(* Logix 5000 project; controller WWTP_SOLIDS_CLX vendor 1 type 14 code 54 rev 17.2; software revision 17.00; part 12 of 16 *)
(* tags used below, declared in another part *)
   Wrk_FirstColdStartT : TIMER;   // Time since first cold start
   Wrk_FirstFailColdT : TIMER;   // Time for cold motor to wait after 1st start failure before ready
   Wrk_SubsFailColdT : TIMER;   // Time for cold motor to wait after 2nd and subs. failures before ready
   Wrk_FirstFailHotT : TIMER;   // Time for hot motor to wait after 1st start failure before ready
   Wrk_SubsFailHotT : TIMER;   // Time for hot motor to wait after 2nd and subs. failures before ready
   Wrk_HotRestartOKT : TIMER;   // Time for hot motor to run so it can restart immediately when stopped
   Wrk_RestartHotT : TIMER;   // Time for hot motor to wait after stop after running less than Hot Restart OK time
   Wrk_HotToColdT : TIMER;   // Time for a stopped hot motor to become cold
   Wrk_State : DINT;   // Instruction State (see state diagram in design docs)
   Wrk_SecondColdStartT : TIMER;   // Time since second cold start
(* P_ResInh, continued *)

ROUTINE Prescan   (* ladder *)
// Clear timers and set to known state
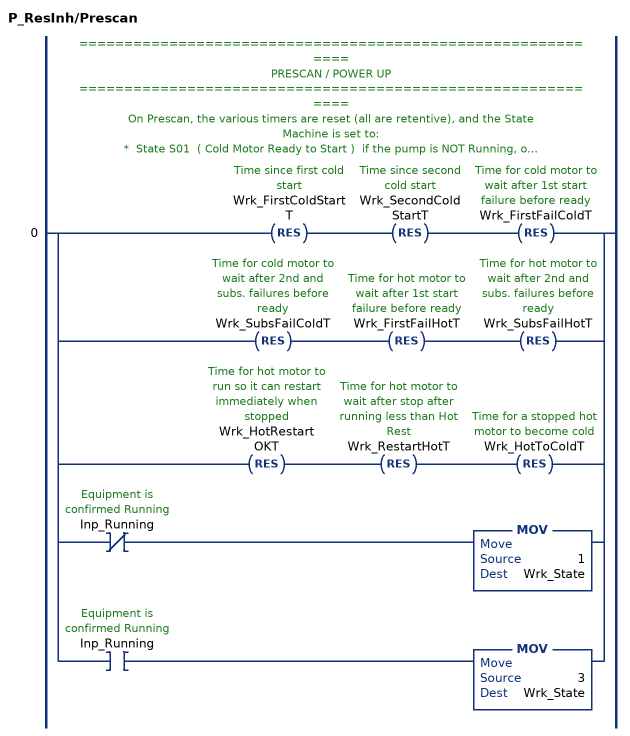
   // ============================================================
   // PRESCAN / POWER UP
   // ============================================================
   // On Prescan, the various timers are reset (all are retentive), and the State
   // Machine is set to:
   // *  State S01  ( Cold Motor Ready to Start )  if the pump is NOT Running, or
   // *  State S03  ( Cold Motor Running )  if the pump is Running.
   0: [RES(Wrk_FirstColdStartT) RES(Wrk_SecondColdStartT) RES(Wrk_FirstFailColdT) ,RES(Wrk_SubsFailColdT) RES(Wrk_FirstFailHotT) RES(Wrk_SubsFailHotT) ,RES(Wrk_HotRestartOKT) RES(Wrk_RestartHotT) RES(Wrk_HotToColdT) ,XIO(Inp_Running) MOV(1,Wrk_State) ,XIC(Inp_Running) MOV(3,Wrk_State) ];
END_ROUTINE
END_ADD_ON_INSTRUCTION

ADD_ON_INSTRUCTION P_RunTime   (* revision 0.7, ExecutePrescan, ExecuteEnableInFalse *)
// Run Time and Starts
// Revision note:
// Aligned name, description and local STRING values, sizes, across instructions.
// Help:
// This Instruction monitors the "Running" and "Starting" Status of a motor or other device and  provides:
// *  Total accumulated run time, in 1/10 hour increments (hour meter)
// *  Total number of starts or start attemptes (count)
// *  Maximum continuous run time for any start (hours)
// *  Program and Maintenance Commands to allow clearing of the totals/maximum
VAR_INPUT
   Inp_Starting : BOOL; {visible}   // 1=Motor is Starting (from motor instruction)
   Inp_Running : BOOL := 1; {visible}   // 1=Motor is Running (from motor instruction)
   Cfg_PCmdClear : BOOL := 1;   // 1=Clear Program Commands on receipt 0=Leave Set
   PCmd_ClearStarts : BOOL;   // Program Command to Clear Count of Starts (attempts)
   PCmd_ClearMaxHrs : BOOL;   // Program Command to Clear Maximum (continuous) Run Time for any start
   PCmd_ClearTotHrs : BOOL;   // Program Command to Clear Total Running Time
   MCmd_ClearStarts : BOOL;   // Maintenance Command to Clear Count of Starts (attempts)
   MCmd_ClearMaxHrs : BOOL;   // Maintenance Command to Clear Maximum (continuous) Run Time for any start
   MCmd_ClearTotHrs : BOOL;   // Maintenance Command to Clear Total Running Time
END_VAR
VAR_OUTPUT
   Val_Starts : DINT; {visible}   // Total number of motor starts or attempts
   Val_CurRunHrs : REAL; {visible}   // Current running time this start (hours)
   Val_MaxRunHrs : REAL; {visible}   // Maximum continuous running time for a given start (hours)
   Val_TotRunHrs : REAL; {visible}   // Total accumulated running time (hours)
END_VAR
VAR
   Wrk_CurHours : DINT;   // Whole hours of current run time
   Wrk_CurRunT : TIMER := (PRE := 2147483647);   // Timer for timing current run time
   Wrk_TotTenths : DINT;   // Tenths of hours of total run time
   Wrk_Starts : COUNTER := (PRE := 2147483647);   // Counter for counting motor starts
   Wrk_TotRunT : TIMER := (PRE := 2147483647);   // Retentive timer for timing 0.1 hour total run time
   Wrk_MaxHours : REAL;   // Internal Maximum Run Hours
END_VAR

ROUTINE EnableInFalse   (* ladder *)
// False Rung or Enable In False: as if motor is Stopped
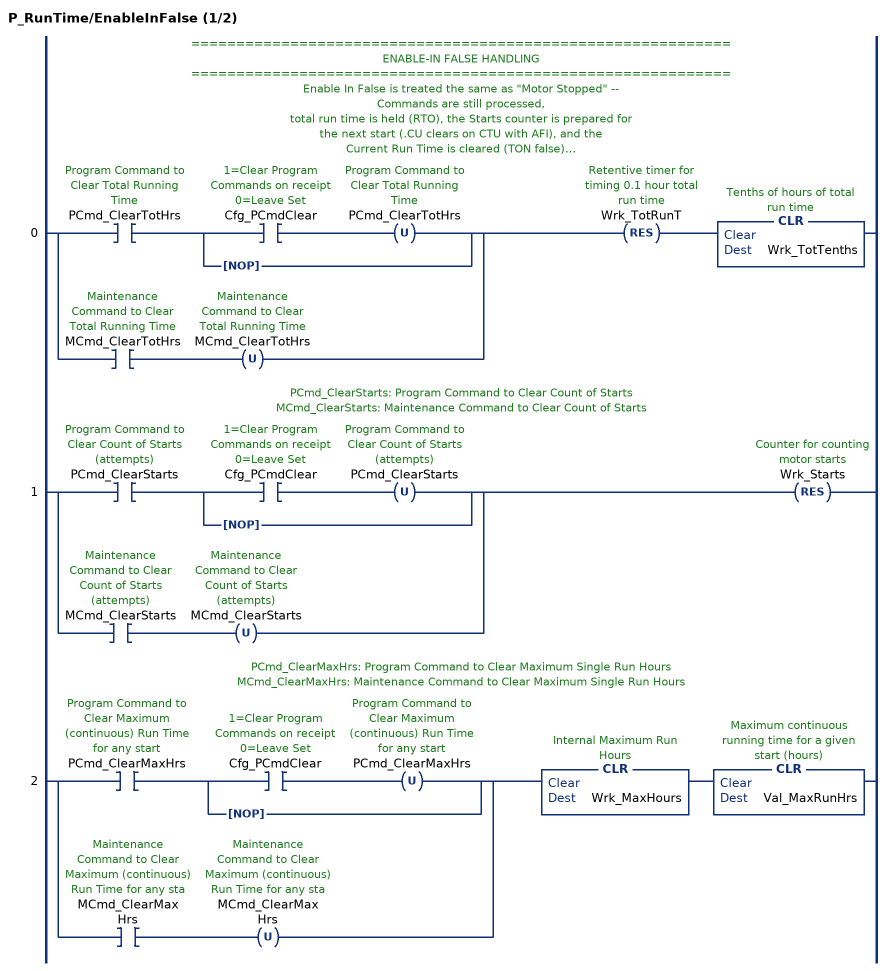
   // ============================================================
   // ENABLE-IN FALSE HANDLING
   // ============================================================
   // Enable In False is treated the same as "Motor Stopped" --
   // Commands are still processed,
   // total run time is held (RTO), the Starts counter is prepared for
   // the next start (.CU clears on CTU with AFI), and the
   // Current Run Time is cleared (TON false).
   // ============================================================
   // COMMAND PROCESSING
   // ============================================================
   // These rungs handle received Commands.  This object has no Modes and
   // Commands are accepted regardless of Mode.  Commands should be
   // restricted to authorized personnel (typically at a maintenance level).
   // PCmd_ClearTotHrs: Program Command to Clear Total Runtime Hours
   // MCmd_ClearTotHrs: Maintenance Command to Clear Total Runtime Hours
   0: [XIC(PCmd_ClearTotHrs) [XIC(Cfg_PCmdClear) OTU(PCmd_ClearTotHrs) ,NOP() ] ,XIC(MCmd_ClearTotHrs) OTU(MCmd_ClearTotHrs) ]RES(Wrk_TotRunT)CLR(Wrk_TotTenths);
   // PCmd_ClearStarts: Program Command to Clear Count of Starts
   // MCmd_ClearStarts: Maintenance Command to Clear Count of Starts
   1: [XIC(PCmd_ClearStarts) [XIC(Cfg_PCmdClear) OTU(PCmd_ClearStarts) ,NOP() ] ,XIC(MCmd_ClearStarts) OTU(MCmd_ClearStarts) ]RES(Wrk_Starts);
   // PCmd_ClearMaxHrs: Program Command to Clear Maximum Single Run Hours
   // MCmd_ClearMaxHrs: Maintenance Command to Clear Maximum Single Run Hours
   2: [XIC(PCmd_ClearMaxHrs) [XIC(Cfg_PCmdClear) OTU(PCmd_ClearMaxHrs) ,NOP() ] ,XIC(MCmd_ClearMaxHrs) OTU(MCmd_ClearMaxHrs) ]CLR(Wrk_MaxHours)CLR(Val_MaxRunHrs);
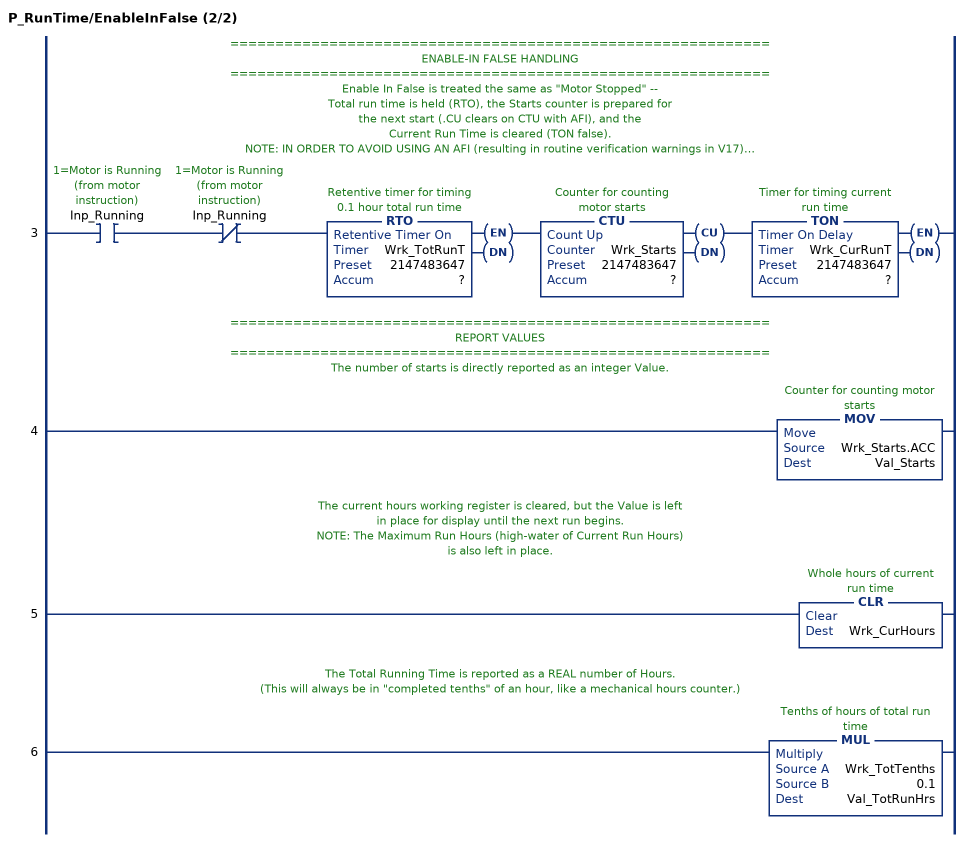
   // ============================================================
   // ENABLE-IN FALSE HANDLING
   // ============================================================
   // Enable In False is treated the same as "Motor Stopped" --
   // Total run time is held (RTO), the Starts counter is prepared for
   // the next start (.CU clears on CTU with AFI), and the
   // Current Run Time is cleared (TON false).
   // NOTE: IN ORDER TO AVOID USING AN AFI (resulting in routine verification warnings in V17),
   // THIS RUNG USES AN XIC AND XIO OF THE SAME BIT TO ENSURE THE
   // TIMERS AND COUNTER ARE SCANNED FALSE.
   // THIS IS NOT DEAD CODE.  IT IS INTENTIONALLY CODED THIS WAY FOR PROPER OPERATION.
   3: XIC(Inp_Running)XIO(Inp_Running)RTO(Wrk_TotRunT,?,?)CTU(Wrk_Starts,?,?)TON(Wrk_CurRunT,?,?);
   // ============================================================
   // REPORT VALUES
   // ============================================================
   // The number of starts is directly reported as an integer Value.
   4: MOV(Wrk_Starts.ACC,Val_Starts);
   // The current hours working register is cleared, but the Value is left
   // in place for display until the next run begins.
   // NOTE: The Maximum Run Hours (high-water of Current Run Hours)
   // is also left in place.
   5: CLR(Wrk_CurHours);
   // The Total Running Time is reported as a REAL number of Hours.
   // (This will always be in "completed tenths" of an hour, like a mechanical hours counter.)
   6: MUL(Wrk_TotTenths,0.1,Val_TotRunHrs);
END_ROUTINE

ROUTINE Logic   (* ladder *)
// Accumulate Run Time (if runnings) and Count Starts
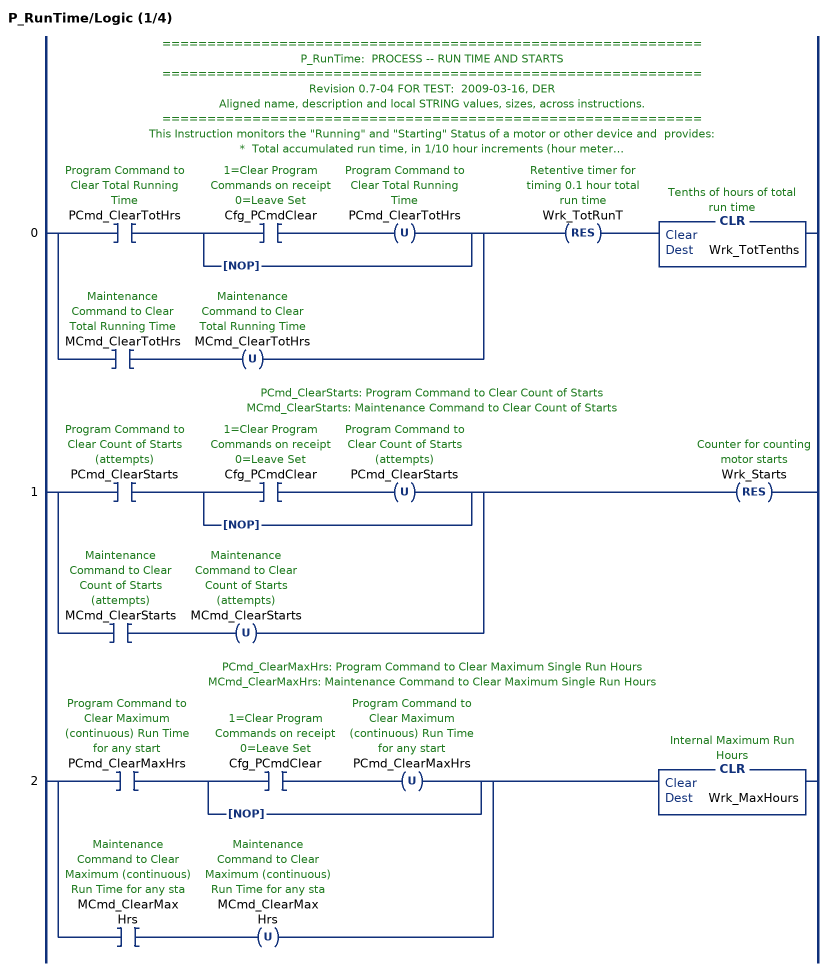
   // ============================================================
   // P_RunTime:  PROCESS -- RUN TIME AND STARTS
   // ============================================================
   // Revision 0.7-04 FOR TEST:  2009-03-16, DER
   // Aligned name, description and local STRING values, sizes, across instructions.
   // ============================================================
   // This Instruction monitors the "Running" and "Starting" Status of a motor or other device and  provides:
   // *  Total accumulated run time, in 1/10 hour increments (hour meter)
   // *  Total number of starts or start attemptes (count)
   // *  Maximum continuous run time for any start (hours)
   // * Commands to allow clearing of the totals/maximum
   // ============================================================
   // COMMAND PROCESSING
   // ============================================================
   // These rungs handle received Commands.  This object has no Modes and
   // Commands are accepted regardless of Mode.  Commands should be
   // restriceted to authorized personnel (typically at a maintenance level).
   // PCmd_ClearTotHrs: Program Command to Clear Total Runtime Hours
   // MCmd_ClearTotHrs: Maintenance Command to Clear Total Runtime Hours
   0: [XIC(PCmd_ClearTotHrs) [XIC(Cfg_PCmdClear) OTU(PCmd_ClearTotHrs) ,NOP() ] ,XIC(MCmd_ClearTotHrs) OTU(MCmd_ClearTotHrs) ]RES(Wrk_TotRunT)CLR(Wrk_TotTenths);
   // PCmd_ClearStarts: Program Command to Clear Count of Starts
   // MCmd_ClearStarts: Maintenance Command to Clear Count of Starts
   1: [XIC(PCmd_ClearStarts) [XIC(Cfg_PCmdClear) OTU(PCmd_ClearStarts) ,NOP() ] ,XIC(MCmd_ClearStarts) OTU(MCmd_ClearStarts) ]RES(Wrk_Starts);
   // PCmd_ClearMaxHrs: Program Command to Clear Maximum Single Run Hours
   // MCmd_ClearMaxHrs: Maintenance Command to Clear Maximum Single Run Hours
   2: [XIC(PCmd_ClearMaxHrs) [XIC(Cfg_PCmdClear) OTU(PCmd_ClearMaxHrs) ,NOP() ] ,XIC(MCmd_ClearMaxHrs) OTU(MCmd_ClearMaxHrs) ]CLR(Wrk_MaxHours);
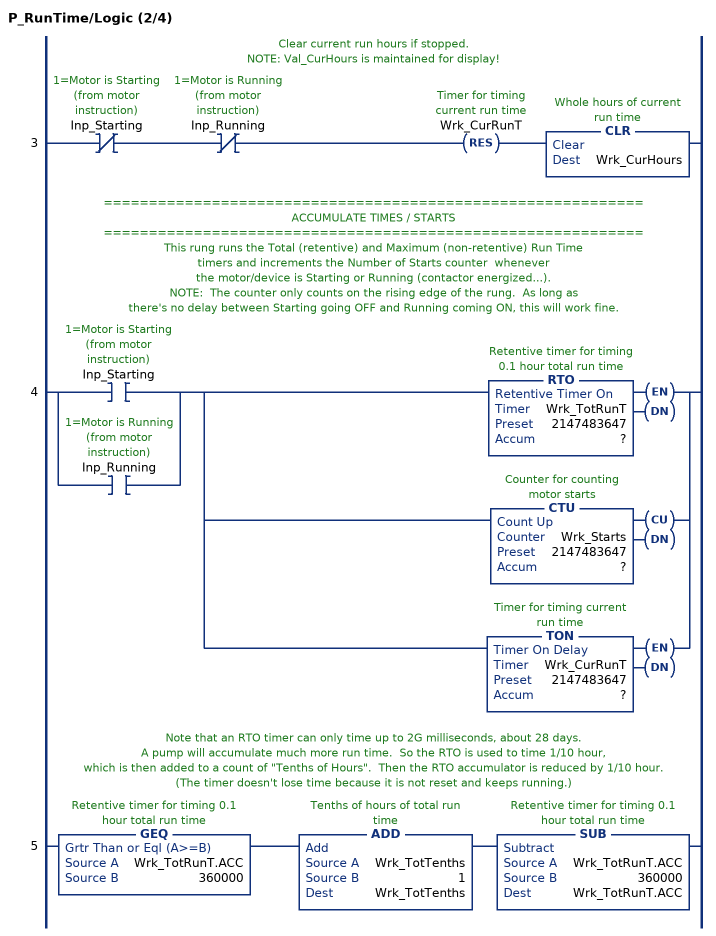
   // Clear current run hours if stopped.
   // NOTE: Val_CurHours is maintained for display!
   3: XIO(Inp_Starting)XIO(Inp_Running)RES(Wrk_CurRunT)CLR(Wrk_CurHours);
   // ============================================================
   // ACCUMULATE TIMES / STARTS
   // ============================================================
   // This rung runs the Total (retentive) and Maximum (non-retentive) Run Time
   // timers and increments the Number of Starts counter  whenever
   //  the motor/device is Starting or Running (contactor energized...).
   // NOTE:  The counter only counts on the rising edge of the rung.  As long as
   // there's no delay between Starting going OFF and Running coming ON, this will work fine.
   4: [XIC(Inp_Starting) ,XIC(Inp_Running) ][RTO(Wrk_TotRunT,?,?) ,CTU(Wrk_Starts,?,?) ,TON(Wrk_CurRunT,?,?) ];
   // Note that an RTO timer can only time up to 2G milliseconds, about 28 days.
   // A pump will accumulate much more run time.  So the RTO is used to time 1/10 hour,
   // which is then added to a count of "Tenths of Hours".  Then the RTO accumulator is reduced by 1/10 hour.
   // (The timer doesn't lose time because it is not reset and keeps running.)
   5: GEQ(Wrk_TotRunT.ACC,360000)ADD(Wrk_TotTenths,1,Wrk_TotTenths)SUB(Wrk_TotRunT.ACC,360000,Wrk_TotRunT.ACC);
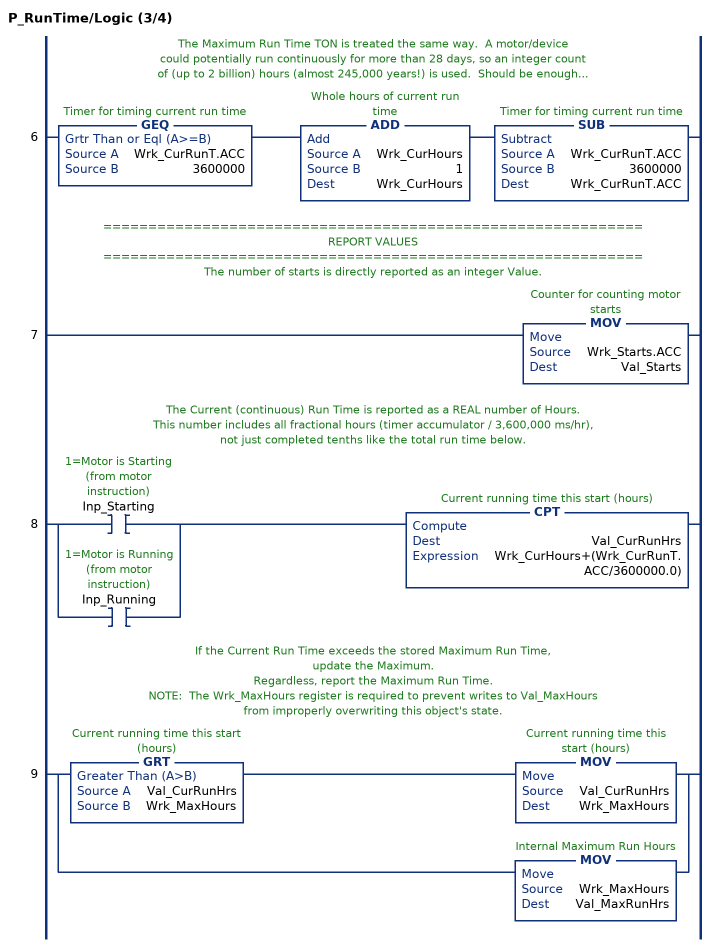
   // The Maximum Run Time TON is treated the same way.  A motor/device
   // could potentially run continuously for more than 28 days, so an integer count
   // of (up to 2 billion) hours (almost 245,000 years!) is used.  Should be enough...
   6: GEQ(Wrk_CurRunT.ACC,3600000)ADD(Wrk_CurHours,1,Wrk_CurHours)SUB(Wrk_CurRunT.ACC,3600000,Wrk_CurRunT.ACC);
   // ============================================================
   // REPORT VALUES
   // ============================================================
   // The number of starts is directly reported as an integer Value.
   7: MOV(Wrk_Starts.ACC,Val_Starts);
   // The Current (continuous) Run Time is reported as a REAL number of Hours.
   // This number includes all fractional hours (timer accumulator / 3,600,000 ms/hr),
   // not just completed tenths like the total run time below.
   8: [XIC(Inp_Starting) ,XIC(Inp_Running) ]CPT(Val_CurRunHrs,Wrk_CurHours+(Wrk_CurRunT.ACC/3600000.0));
   // If the Current Run Time exceeds the stored Maximum Run Time,
   // update the Maximum.
   // Regardless, report the Maximum Run Time.
   // NOTE:  The Wrk_MaxHours register is required to prevent writes to Val_MaxHours
   // from improperly overwriting this object's state.
   9: [GRT(Val_CurRunHrs,Wrk_MaxHours) MOV(Val_CurRunHrs,Wrk_MaxHours) ,MOV(Wrk_MaxHours,Val_MaxRunHrs) ];
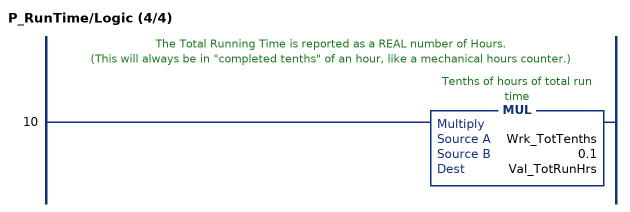
   // The Total Running Time is reported as a REAL number of Hours.
   // (This will always be in "completed tenths" of an hour, like a mechanical hours counter.)
   10: MUL(Wrk_TotTenths,0.1,Val_TotRunHrs);
END_ROUTINE

ROUTINE Prescan   (* ladder *)
// Set Current Run time internally to 0.  Display value is left in place.
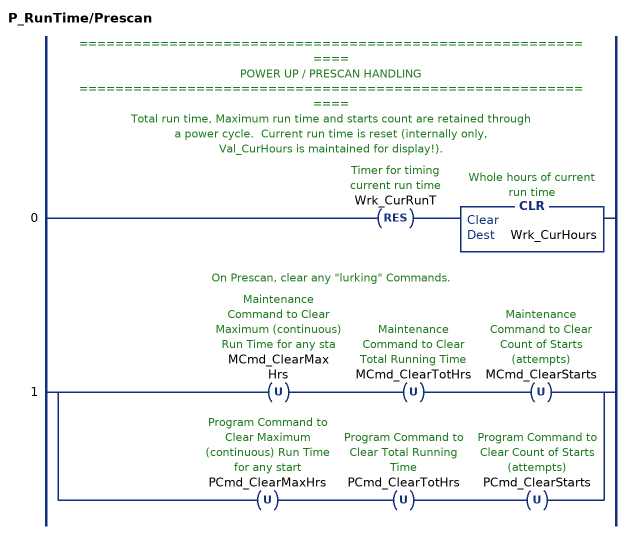
   // ============================================================
   // POWER UP / PRESCAN HANDLING
   // ============================================================
   // Total run time, Maximum run time and starts count are retained through
   // a power cycle.  Current run time is reset (internally only,
   // Val_CurHours is maintained for display!).
   0: RES(Wrk_CurRunT)CLR(Wrk_CurHours);
   // On Prescan, clear any "lurking" Commands.
   1: [OTU(MCmd_ClearMaxHrs) OTU(MCmd_ClearTotHrs) OTU(MCmd_ClearStarts) ,OTU(PCmd_ClearMaxHrs) OTU(PCmd_ClearTotHrs) OTU(PCmd_ClearStarts) ];
END_ROUTINE
END_ADD_ON_INSTRUCTION

ADD_ON_INSTRUCTION P_ValveMO   (* revision 0.9, ExecutePrescan, ExecuteEnableInFalse *)
// Motor Operated Valve
// Revision note:
// Aligned name, description and local STRING values, sizes, across instructions.
// Help:
// This Instruction controls and monitors a motor-operated
// valve (typ. two position: opened, closed) and provides:
// *  Ability to command valve to open, command valve to close, and,
//      optionally, command valve to stop motion (operator only)
// *  Ability to reverse valve travel (for valves with the ability to accept a Stop output)
// *  Monitoring of limit switch feedback, display of actual valve status
// *  Detection of failure to move (full stall), failure to reach position (transit stall)
// *  Monitoring of Permissive conditions to motor the valve open, and separate
//      Permissive conditions to motor the valve closed
// *  Simulation, providing feedback of a working valve while disabling outputs
// *  Monitoring of I/O communication faults
// *  Alarms for Full Stall, Transit Stall, Actuator Failure (separate input), I/O Fault
// *  Operation in Hand, Maintenance, Override, Program and Operator Modes
// *  "Available" status for use by automation logic to know whether valve
//      can be controlled by other objects.
VAR_INPUT
   Inp_OpenLS : BOOL; {visible}   // Valve Open Limit Switch 1=confirmed OPEN
   Inp_ClosedLS : BOOL; {visible}   // Valve Closed Limit Switch 1=confirmed CLOSED
   Inp_ActuatorFault : BOOL; {visible}   // Valve Actuator Fault (overload, etc.), 0=OK, 1=Fault)
   Inp_OpenPermOK : BOOL := 1; {visible}   // 1=Open Permissives OK, Valve can motor open
   Inp_OpenNBPermOK : BOOL := 1; {visible}   // 1=Non-Bypassable Open Permissives OK, valve can motor open
   Inp_ClosePermOK : BOOL := 1; {visible}   // 1=Close Permissives OK, Valve can motor closed
   Inp_CloseNBPermOK : BOOL := 1; {visible}   // 1=Non-Bypassable Close Permissives OK, valve can motor closed
   Inp_IOFault : BOOL;   // Input Communication Status 0=OK, 1=fail
   Inp_Sim : BOOL;   // 1=Simulate working valve; 0=Open/Close/ Monitor actual valve
   Inp_Hand : BOOL; {visible}   // 1=Select Hand (hardwired) Mode
   Inp_Ovrd : BOOL; {visible}   // 1=Select Override Mode
   Inp_OvrdOpen : BOOL; {visible}   // 1=Override to OPEN, 0=do not override open
   Inp_OvrdClose : BOOL; {visible}   // 1=Override to CLOSED, 0=do not override closed
   Inp_OvrdStop : BOOL;   // 1=Override to STOP moving, 0=do not override to STOP
   Inp_Reset : BOOL; {visible}   // 1=Reset all fault conditions and latched Alarms
   Cfg_HasOpenLS : BOOL;   // 1=Valve provides an Open Limit Switch signal
   Cfg_HasClosedLS : BOOL;   // 1=Valve provides a Closed Limit Switch signal
   Cfg_UseOpenLS : BOOL;   // 1=Valve Open LS should be used for failure checking
   Cfg_UseClosedLS : BOOL;   // 1=Valve Closed LS should be used for failure checking
   Cfg_LSFail : BOOL := 1;   // 1=both switches ON=fail, 0=both switches OFF=fail
   Cfg_HasStop : BOOL;   // 1=Stop output can be used to break local seal-in and stop valve motion
   Cfg_HasOpenPermObj : BOOL;   // 1=Tells HMI a P_Perm is connected to Inp_OpenPermOK
   Cfg_HasClosePermObj : BOOL;   // 1=Tells HMI a P_Perm is connected to Inp_ClosePermOK
   Cfg_PCmdClear : BOOL := 1;   // 1=Clear Program Commands on receipt 0=Leave Set
   Cfg_OvrdPerm : BOOL;   // 1=Override ignores Bypassable Perm; 0=always use Perm
   Cfg_HasFullStallAlm : BOOL;   // 1=Full Stall Alarm exists and will be checked
   Cfg_HasTransitStallAlm : BOOL;   // 1=Transit Stall Alarm exists and will be checked
   Cfg_HasActuatorFaultAlm : BOOL;   // 1=Actuator Fault Alarm exists and will be checked
   Cfg_HasIOFaultAlm : BOOL;   // 1=I/O Fault Alarm exists and will be checked
   Cfg_FullStallResetReqd : BOOL;   // 1=Reset requied to clear Full Stall Alarm
   Cfg_TransitStallResetReqd : BOOL;   // 1=Reset required to clear Transit Stall Alarm
   Cfg_ActuatorFaultResetReqd : BOOL;   // 1=Reset required to clear Actuator Fault Alarm
   Cfg_IOFaultResetReqd : BOOL;   // 1=Reset required to clear I/O Fault Alarm
   Cfg_FullStallAckReqd : BOOL := 1;   // 1=Acknowledge required for Full Stall Alarm
   Cfg_TransitStallAckReqd : BOOL := 1;   // 1=Acknowledge required for Transit Stall Alarm
   Cfg_ActuatorFaultAckReqd : BOOL := 1;   // 1=Acknowledge required for Actuator Fault Alarm
   Cfg_IOFaultAckReqd : BOOL := 1;   // 1=Acknowledge required for I/O Fault Alarm
   Cfg_FullStallSeverity : SINT := 4;   // Full Stall Alarm Severity 1=info 2=warn 3=excep 4=fault
   Cfg_TransitStallSeverity : SINT := 4;   // Transit Stall Alarm Severity 1=info 2=warn 3=excep 4=fault
   Cfg_ActuatorFaultSeverity : SINT := 2;   // Actuator Fault Alarm Severity 1=info 2=warn 3=excep 4=fault
   Cfg_IOFaultSeverity : SINT := 4;   // I/O Fault Alarm Severity 1=info 2=warn 3=excep 4=fault
   Cfg_OutPulseT : DINT := 5;   // Time (in seconds) to pulse valve outputs (0 = outputs maintained ON)
   Cfg_SimFdbkT : DINT := 20;   // Delay to echo back of Open/Closed status when in Simulation (sec)
   Cfg_FullStallT : DINT := 15;   // After commanded, time with no motion before Fault (sec)
   Cfg_TransitStallT : DINT := 60;   // After command, time to reach position before fault (sec)
   PSet_Owner : DINT;   // Program Owner Request ID (non-zero) or Release (zero)
   PCmd_Open : BOOL;   // Program Command to Open Valve
   PCmd_Close : BOOL;   // Program Command to Close Valve
   PCmd_Acq : BOOL;   // Program Command to Acquire ownership (Oper/OOS to Prog)
   PCmd_Rel : BOOL;   // Program Command to Release ownership (Prog to OOS)
   PCmd_Lock : BOOL;   // Program Command to Lock Mode in Prog
   PCmd_Unlock : BOOL;   // Program Command to Unlock Mode
   PCmd_Reset : BOOL;   // Program Command to Reset all Alarms requiring Reset
   PCmd_FullStallAck : BOOL;   // Program Command to Acknowledge Full Stall Alarm
   PCmd_FullStallInhibit : BOOL;   // Program Command to Inhibit Full Stall Alarm
   PCmd_FullStallUninhibit : BOOL;   // Program Command to Uninhibit Full Stall Alarm
   PCmd_TransitStallAck : BOOL;   // Program Command to Acknowledge Transit Stall Alarm
   PCmd_TransitStallInhibit : BOOL;   // Program Command to Inhibit Transit Stall Alarm
   PCmd_TransitStallUninhibit : BOOL;   // Program Command to Uninhibit Transit Stall Alarm
   PCmd_ActuatorFaultAck : BOOL;   // Program Command to Acknowledge Actuator Fault Alarm
   PCmd_ActuatorFaultInhibit : BOOL;   // Program Command to Inhibit Actuator Fault Alarm
   PCmd_ActuatorFaultUninhibit : BOOL;   // Program Command to Uninhibit Actuator Fault Alarm
   PCmd_IOFaultAck : BOOL;   // Program Command to Acknowledge I/O Fault Alarm
   PCmd_IOFaultInhibit : BOOL;   // Program Command to Inhibit I/O Fault Alarm
   PCmd_IOFaultUninhibit : BOOL;   // Program Command to Uninhibit I/O Fault Alarm
   OCmd_Open : BOOL;   // Operator Command to Open Valve
   OCmd_Close : BOOL;   // Operator Command to Close Valve
   OCmd_Stop : BOOL;   // Operator Command to Stop Valve Motion
   OCmd_Bypass : BOOL;   // Operator Command to Bypass all Bypassable Interlocks and Permissives
   OCmd_Check : BOOL;   // Operator Command to Check (not bypass) all Interlocks and Permissives
   MCmd_Disable : BOOL;   // Maintenance Command to Disable Valve
   MCmd_Enable : BOOL;   // Maintenance Command to Enable (allow to energize) Valve
   OCmd_Reset : BOOL;   // Operator Command to Reset all Alarms requiring Reset
END_VAR
VAR_OUTPUT
   Out_Open : BOOL; {visible}   // 1=Run actuator motor to OPEN Valve
   Out_Close : BOOL; {visible}   // 1=Run actuator motor to CLOSE Valve
   Out_Stop : BOOL;   // 1=Break seal-in circuit in actuator to STOP Valve motion
   Val_Owner : DINT;   // Current Object Owner ID (0=not owned)
   Val_Notify : SINT;   // Current Alarm Level and Acknowledgement (enumeration)
   Sts_Closed : BOOL; {visible}   // 1=Valve requested to Close and is confirmed Closed
   Sts_CmdToOpen : BOOL; {visible}   // 1=Valve commanded to Open, has not yet moved off Open LS
   Sts_Opening : BOOL; {visible}   // 1=Valve requested to open and awaiting open feedback
   Sts_Opened : BOOL; {visible}   // 1=Valve requested to open and is confirmed Opened
   Sts_CmdToClose : BOOL; {visible}   // 1=Valve commanded to Close, has not yet moved off Closed LS
   Sts_Closing : BOOL; {visible}   // 1=Valve requested to Close and awaiting Closed feedback
   Sts_Stopped : BOOL;   // 1=Valve requested to Stop and is not at either end of travel
   Sts_Available : BOOL;   // 1=Valve available for control by automation (Prog)
   Sts_Bypass : BOOL;   // 1=Bypassable Interlocks and Permissives are Bypassed
   Sts_Disabled : BOOL;   // 1=Valve is Disabled
   Sts_LSFail : BOOL;   // 1=Limit Switch Overlap Failure
   Sts_Err : BOOL; {visible}   // 1=Error in Config: see detail bits for reason
   Err_Timer : BOOL;   // 1=Error in Config: Invalid Check or Pulse Time (use 0 to 2147483)
   Err_Sim : BOOL;   // 1=Error in Config: Simulation timer preset (use 0 to 2147483)
   Err_Alarm : BOOL;   // 1=Error in Config: Invalid Alarm Severity
   Sts_Hand : BOOL; {visible}   // 1=Mode is Hand (supersedes Maint, Ovrd, Prog, Oper)
   Sts_Maint : BOOL; {visible}   // 1=Mode is Maintenance (supersedes Ovrd, Prog, Oper)
   Sts_Ovrd : BOOL; {visible}   // 1=Mode is Override (supersedes Prog, Oper)
   Sts_Prog : BOOL; {visible}   // 1=Mode is Program (auto)
   Sts_Oper : BOOL := 1; {visible}   // 1=Mode is Operator (manual)
   Sts_ProgOperLock : BOOL;   // 1=Program or Operator has requested Mode Lock
   Sts_FullStall : BOOL;   // 1=Valve Full Stall (failed to move at all) (One-Shot)
   Alm_FullStall : BOOL;   // 1=Valve Full Stall (failed to move at all) Alarm
   Ack_FullStall : BOOL;   // 1=Full Stall Alarm has been acknowledged
   Sts_FullStallDisabled : BOOL;   // 1=Full Stall Alarm has been disabled (will not be sent)
   Sts_FullStallInhibited : BOOL;   // 1=Full Stall Alarm has been inhibited by logic
   Sts_FullStallSuppressed : BOOL;   // 1=Full Stall Alarm has been suppressed (logged only)
   Sts_TransitStall : BOOL;   // 1=Valve Transit Stall (did not reach target position) (One-Shot)
   Alm_TransitStall : BOOL;   // 1=Valve Transit Stall (did not reach target pos.) Alarm
   Ack_TransitStall : BOOL;   // 1=Transit Stall Alarm has been acknowledged
   Sts_TransitStallDisabled : BOOL;   // 1=Transit Stall Alarm has been disabled (will not be sent)
   Sts_TransitStallInhibited : BOOL;   // 1=Transit Stall Alarm has been inhibited by logic
   Sts_TransitStallSuppressed : BOOL;   // 1=Transit Stall Alarm has been suppressed (logged only)
   Sts_ActuatorFault : BOOL;   // 1=Actuator Fault detected (input)
   Alm_ActuatorFault : BOOL;   // 1=Alarm: Actuator Fault Detected
   Ack_ActuatorFault : BOOL;   // 1=Actuator Fault Alarm has been acknowledged
   Sts_ActuatorFaultDisabled : BOOL;   // 1=Actuator Fault Alarm is Disabled (not saved or sent)
   Sts_ActuatorFaultInhibited : BOOL;   // 1=Actuator Fault Alarm has been inhibited by logic
   Sts_ActuatorFaultSuppressed : BOOL;   // 1=Actuator Fault Alarm has been suppressed (logged only)
   Sts_IOFault : BOOL;   // I/O Comm Fault Status (0=OK, 1=Bad)
   Alm_IOFault : BOOL;   // 1=I/O Fault Alarm
   Ack_IOFault : BOOL;   // 1=I/O Fault Alarm has been acknowledged
   Sts_IOFaultDisabled : BOOL;   // 1=I/O Fault Alarm is Disabled (not saved or sent)
   Sts_IOFaultInhibited : BOOL;   // 1=I/O Fault Alarm has been inhibited by logic
   Sts_IOFaultSuppressed : BOOL;   // 1=I/O Fault Alarm has been suppressed (logged only)
   Rdy_Open : BOOL;   // 1=Ready to receive OCmd_Open (enables HMI button)
   Rdy_Close : BOOL;   // 1=Ready to receive OCmd_Close (enables HMI button)
   Rdy_Stop : BOOL;   // 1=Ready to receive OCmd_Stop (enables HMI button)
   Rdy_Bypass : BOOL;   // 1=Ready to receive OCmd_Bypass (enables HMI button)
   Rdy_Check : BOOL;   // 1=Ready to receive OCmd_Check (enables HMI button)
   Rdy_Disable : BOOL;   // 1=Ready to receive MCmd_Disable (enables HMI button)
   Rdy_Enable : BOOL;   // 1=Ready to receive MCmd_Enable (enables HMI button)
   Rdy_Reset : BOOL;   // 1=Ready to receive OCmd_Reset (enables HMI button)
END_VAR
VAR
   Mode : P_Mode := (Cfg_PCmdClear := 1, Cfg_OvrdOverLock := 1, Sts_Oper := 1, Rdy_Rel := 1, Rdy_AcqLock := 1);   // Valve Mode Selection
   IOFault : P_Alarm := (Inp := 1, Cfg_AckReqd := 1, Cfg_Severity := 3, Ack := 1, Rdy_Disable := 1);   // I/O Fault Alarm
   ActuatorFault : P_Alarm := (Inp := 1, Cfg_AckReqd := 1, Cfg_Severity := 3, Ack := 1, Rdy_Disable := 1);   // Actuator Fault Alarm
   TransitStall : P_Alarm := (Inp := 1, Cfg_AckReqd := 1, Cfg_Severity := 3, Ack := 1, Rdy_Disable := 1);   // Valve Transit Stall (moved but did not reach target) Alarm
   FullStall : P_Alarm := (Inp := 1, Cfg_AckReqd := 1, Cfg_Severity := 3, Ack := 1, Rdy_Disable := 1);   // Valve Full Stall (did not move) Alarm
   Cfg_Tag : STRING_20 := 'P_ValveMO';   // Tagname for display on HMI
   Cfg_Label : STRING_20 := 'Valve Control';   // Label for graphic symbol displayed on HMI
   Cfg_Desc : STRING_40 := 'Motor Operated Valve';   // Description for display on HMI
   Wrk_Open : BOOL;   // 1=Requested to OPEN Valve
   Wrk_SimOpenT : TIMER;   // Simulation Delay until Opened
   Wrk_Fault : BOOL;   // 1=a Valve Fault has been detected
   Wrk_SimCloseT : TIMER;   // Simulation Delay until Closed
   Wrk_OpenFdbk : BOOL;   // 1=LS Feedback shows valve confirmed open
   Wrk_Notify : DINT;   // Buffer for building Val_Notify
   Wrk_Bypass : BOOL;   // Internal Bypassable Permissives and Interlocks are Bypassed flag
   Wrk_Disabled : BOOL;   // Internal Valve is Disabled
   Wrk_ClosedFdbk : BOOL;   // 1=LS Feedback shows valve confirmed closed
   Wrk_LSFailFdbk : BOOL;   // 1=LS Feedback shows Limit Switch Failure
   Wrk_TravelFdbk : BOOL;   // 1=LS Feedback shows Valve is Traveling
   Wrk_Stop : BOOL;   // 1=Requested to STOP Valve
   Wrk_Close : BOOL;   // 1-Requested to CLOSE Valve
   Wrk_StopPulseT : TIMER;   // Timer for Out_Stop pulse time
   Wrk_ClosePulseT : TIMER;   // Timer for Out_Close pulse time
   Wrk_OpenPulseT : TIMER;   // Timer for Out_Open pulse time
   Wrk_TransitStallT : TIMER;   // Timer for Transit Stall Check
   Wrk_FullStallT : TIMER;   // Timer for Full Stall Check
END_VAR

ROUTINE EnableInFalse   (* ladder *)
// Disabled is asserted; Outputs OFF; Valve Status shown but Alarms disabled
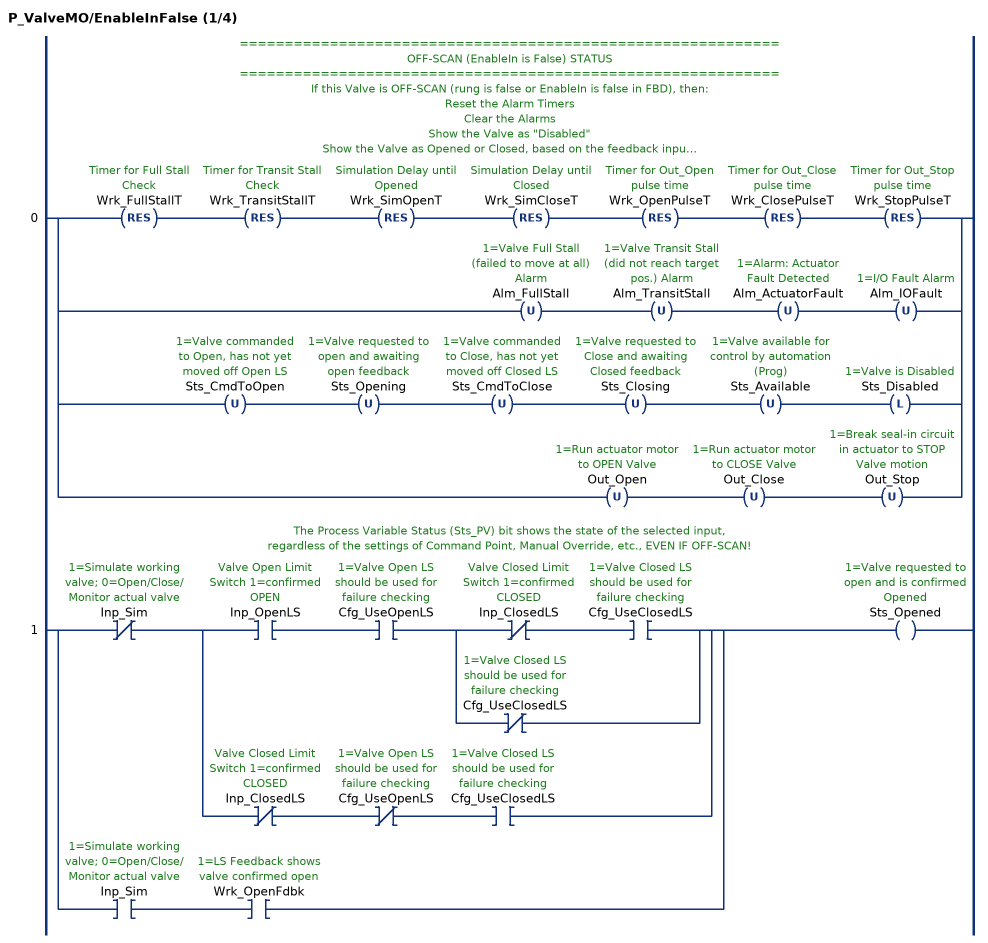
   // ============================================================
   // OFF-SCAN (EnableIn is False) STATUS
   // ============================================================
   // If this Valve is OFF-SCAN (rung is false or EnableIn is false in FBD), then:
   // Reset the Alarm Timers
   // Clear the Alarms
   // Show the Valve as "Disabled"
   // Show the Valve as Opened or Closed, based on the feedback input
   // Turn off the Outputs
   // Other data are left in Last State!
   0: [RES(Wrk_FullStallT) RES(Wrk_TransitStallT) RES(Wrk_SimOpenT) RES(Wrk_SimCloseT) RES(Wrk_OpenPulseT) RES(Wrk_ClosePulseT) RES(Wrk_StopPulseT) ,OTU(Alm_FullStall) OTU(Alm_TransitStall) OTU(Alm_ActuatorFault) OTU(Alm_IOFault) ,OTU(Sts_CmdToOpen) OTU(Sts_Opening) OTU(Sts_CmdToClose) OTU(Sts_Closing) OTU(Sts_Available) OTL(Sts_Disabled) ,OTU(Out_Open) OTU(Out_Close) OTU(Out_Stop) ];
   // The Process Variable Status (Sts_PV) bit shows the state of the selected input,
   // regardless of the settings of Command Point, Manual Override, etc., EVEN IF OFF-SCAN!
   1: [XIO(Inp_Sim) [XIC(Inp_OpenLS) XIC(Cfg_UseOpenLS) [XIO(Inp_ClosedLS) XIC(Cfg_UseClosedLS) ,XIO(Cfg_UseClosedLS) ] ,XIO(Inp_ClosedLS) XIO(Cfg_UseOpenLS) XIC(Cfg_UseClosedLS) ] ,XIC(Inp_Sim) XIC(Wrk_OpenFdbk) ]OTE(Sts_Opened);
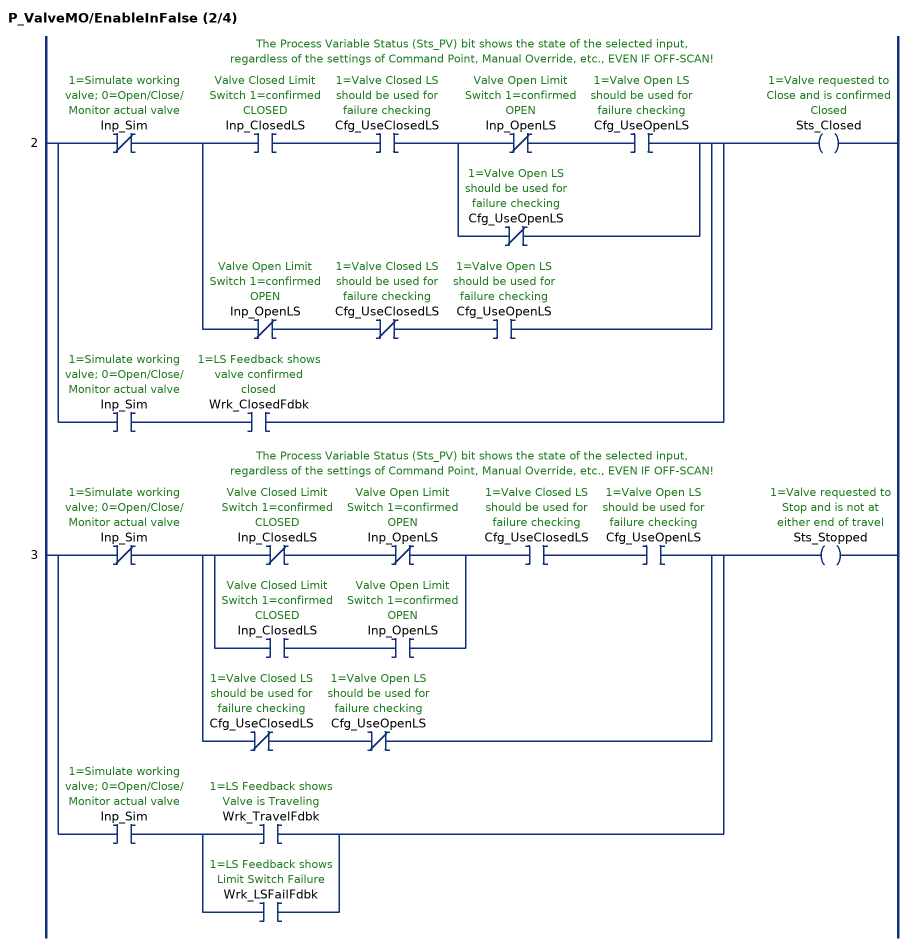
   // The Process Variable Status (Sts_PV) bit shows the state of the selected input,
   // regardless of the settings of Command Point, Manual Override, etc., EVEN IF OFF-SCAN!
   2: [XIO(Inp_Sim) [XIC(Inp_ClosedLS) XIC(Cfg_UseClosedLS) [XIO(Inp_OpenLS) XIC(Cfg_UseOpenLS) ,XIO(Cfg_UseOpenLS) ] ,XIO(Inp_OpenLS) XIO(Cfg_UseClosedLS) XIC(Cfg_UseOpenLS) ] ,XIC(Inp_Sim) XIC(Wrk_ClosedFdbk) ]OTE(Sts_Closed);
   // The Process Variable Status (Sts_PV) bit shows the state of the selected input,
   // regardless of the settings of Command Point, Manual Override, etc., EVEN IF OFF-SCAN!
   3: [XIO(Inp_Sim) [[XIO(Inp_ClosedLS) XIO(Inp_OpenLS) ,XIC(Inp_ClosedLS) XIC(Inp_OpenLS) ] XIC(Cfg_UseClosedLS) XIC(Cfg_UseOpenLS) ,XIO(Cfg_UseClosedLS) XIO(Cfg_UseOpenLS) ] ,XIC(Inp_Sim) [XIC(Wrk_TravelFdbk) ,XIC(Wrk_LSFailFdbk) ] ]OTE(Sts_Stopped);
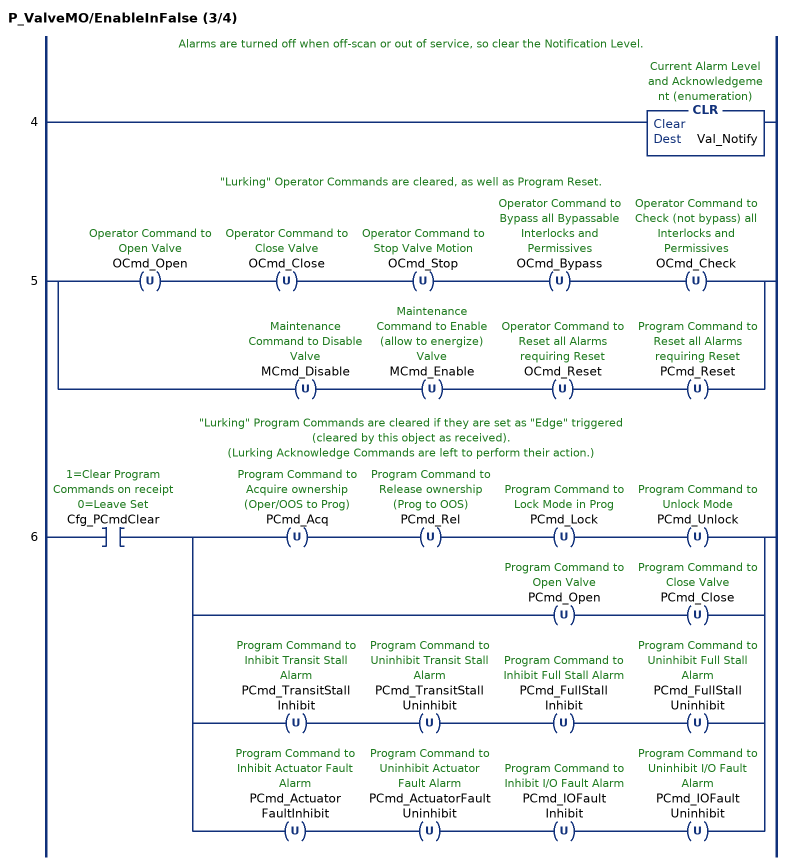
   // Alarms are turned off when off-scan or out of service, so clear the Notification Level.
   4: CLR(Val_Notify);
   // "Lurking" Operator Commands are cleared, as well as Program Reset.
   5: [OTU(OCmd_Open) OTU(OCmd_Close) OTU(OCmd_Stop) OTU(OCmd_Bypass) OTU(OCmd_Check) ,OTU(MCmd_Disable) OTU(MCmd_Enable) OTU(OCmd_Reset) OTU(PCmd_Reset) ];
   // "Lurking" Program Commands are cleared if they are set as "Edge" triggered
   // (cleared by this object as received).
   // (Lurking Acknowledge Commands are left to perform their action.)
   6: XIC(Cfg_PCmdClear)[OTU(PCmd_Acq) OTU(PCmd_Rel) OTU(PCmd_Lock) OTU(PCmd_Unlock) ,OTU(PCmd_Open) OTU(PCmd_Close) ,OTU(PCmd_TransitStallInhibit) OTU(PCmd_TransitStallUninhibit) OTU(PCmd_FullStallInhibit) OTU(PCmd_FullStallUninhibit) ,OTU(PCmd_ActuatorFaultInhibit) OTU(PCmd_ActuatorFaultUninhibit) OTU(PCmd_IOFaultInhibit) OTU(PCmd_IOFaultUninhibit) ];
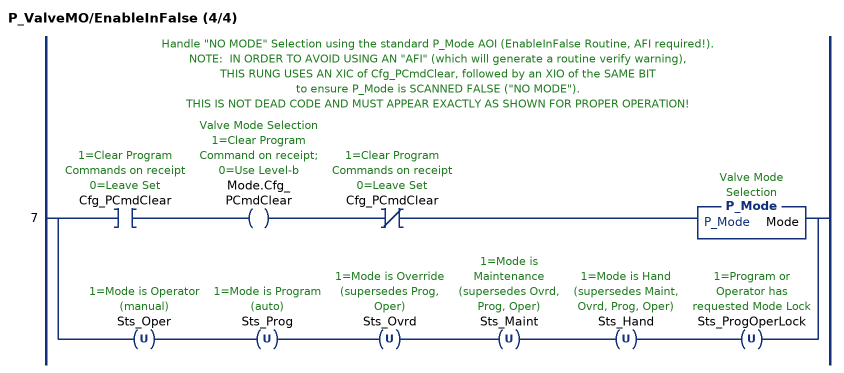
   // Handle "NO MODE" Selection using the standard P_Mode AOI (EnableInFalse Routine, AFI required!).
   // NOTE:  IN ORDER TO AVOID USING AN "AFI" (which will generate a routine verify warning),
   // THIS RUNG USES AN XIC of Cfg_PCmdClear, followed by an XIO of the SAME BIT
   // to ensure P_Mode is SCANNED FALSE ("NO MODE").
   // THIS IS NOT DEAD CODE AND MUST APPEAR EXACTLY AS SHOWN FOR PROPER OPERATION!
   7: [XIC(Cfg_PCmdClear) OTE(Mode.Cfg_PCmdClear) XIO(Cfg_PCmdClear) P_Mode(Mode) ,OTU(Sts_Oper) OTU(Sts_Prog) OTU(Sts_Ovrd) OTU(Sts_Maint) OTU(Sts_Hand) OTU(Sts_ProgOperLock) ];
END_ROUTINE

ROUTINE Logic   (* ladder *)
// Normal Scan: control / monitor solenoid-operated valve
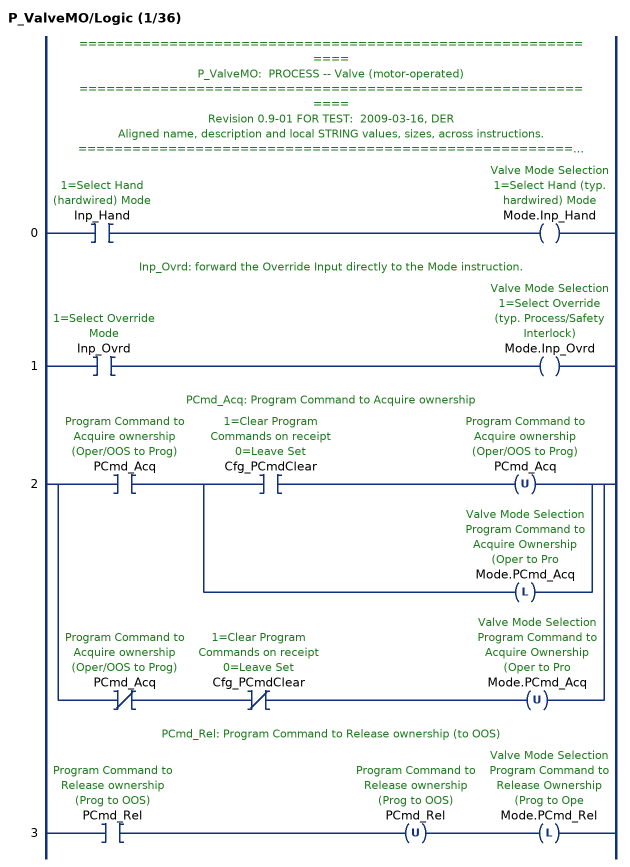
   // ============================================================
   // P_ValveMO:  PROCESS -- Valve (motor-operated)
   // ============================================================
   // Revision 0.9-01 FOR TEST:  2009-03-16, DER
   // Aligned name, description and local STRING values, sizes, across instructions.
   // ============================================================
   // This Instruction controls and monitors a motor-operated
   // valve (typ. two position: opened, closed) and provides:
   // *  Ability to command valve to open, command valve to close, and,
   // optionally, command valve to stop motion (operator only)
   // *  Ability to reverse valve travel (for valves with the ability to accept a Stop output)
   // *  Monitoring of limit switch feedback, display of actual valve status
   // *  Detection of failure to move (full stall), failure to reach position (transit stall)
   // *  Monitoring of Permissive conditions to motor the valve open, and separate
   // Permissive conditions to motor the valve closed
   // *  Simulation, providing feedback of a working valve while disabling outputs
   // *  Monitoring of I/O communication faults
   // *  Alarms for Full Stall, Transit Stall, Actuator Failure (separate input), I/O Fault
   // *  Operation in Hand, Maintenance, Override, Program and Operator Modes
   // *  "Available" status for use by automation logic to know whether valve
   //       can be controlled by other objects.
   // ============================================================
   // POWERUP / INVALID STATE HANDLING
   // ============================================================
   // Mode states are retained through a power cycle.
   // Valve "open" request is set or cleared on first scan; depending on fail state of valve.
   // ============================================================
   // MODE PROCESSING
   // ============================================================
   // These rungs handle received Mode Inputs and Commands:
   // NOTE:  Operator Commands for Mode, Alarm are sent directly to the contained P_Mode and P_Alarm AOIs.
   // Inp_Hand: forward the Hand Input directly to the Mode instruction.
   0: XIC(Inp_Hand)OTE(Mode.Inp_Hand);
   // Inp_Ovrd: forward the Override Input directly to the Mode instruction.
   1: XIC(Inp_Ovrd)OTE(Mode.Inp_Ovrd);
   // PCmd_Acq: Program Command to Acquire ownership
   2: [XIC(PCmd_Acq) [XIC(Cfg_PCmdClear) OTU(PCmd_Acq) ,OTL(Mode.PCmd_Acq) ] ,XIO(PCmd_Acq) XIO(Cfg_PCmdClear) OTU(Mode.PCmd_Acq) ];
   // PCmd_Rel: Program Command to Release ownership (to OOS)
   3: XIC(PCmd_Rel)OTU(PCmd_Rel)OTL(Mode.PCmd_Rel);
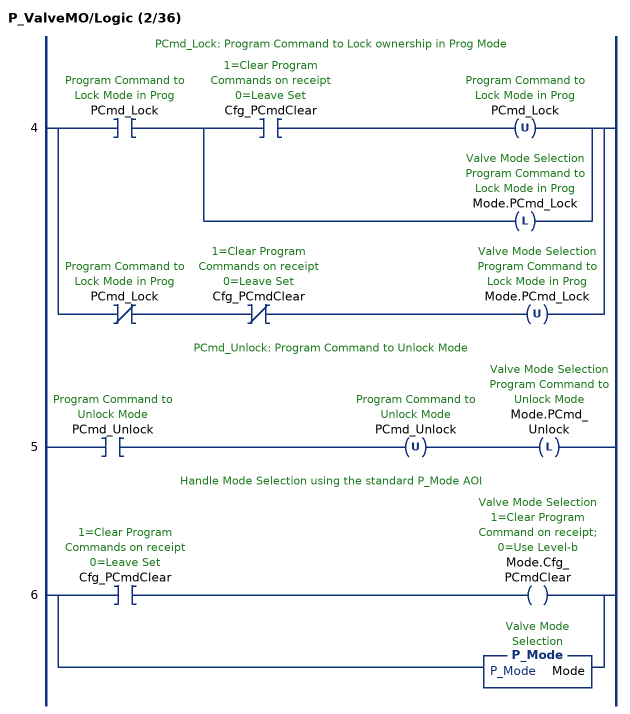
   // PCmd_Lock: Program Command to Lock ownership in Prog Mode
   4: [XIC(PCmd_Lock) [XIC(Cfg_PCmdClear) OTU(PCmd_Lock) ,OTL(Mode.PCmd_Lock) ] ,XIO(PCmd_Lock) XIO(Cfg_PCmdClear) OTU(Mode.PCmd_Lock) ];
   // PCmd_Unlock: Program Command to Unlock Mode
   5: XIC(PCmd_Unlock)OTU(PCmd_Unlock)OTL(Mode.PCmd_Unlock);
   // Handle Mode Selection using the standard P_Mode AOI
   6: [XIC(Cfg_PCmdClear) OTE(Mode.Cfg_PCmdClear) ,P_Mode(Mode) ];
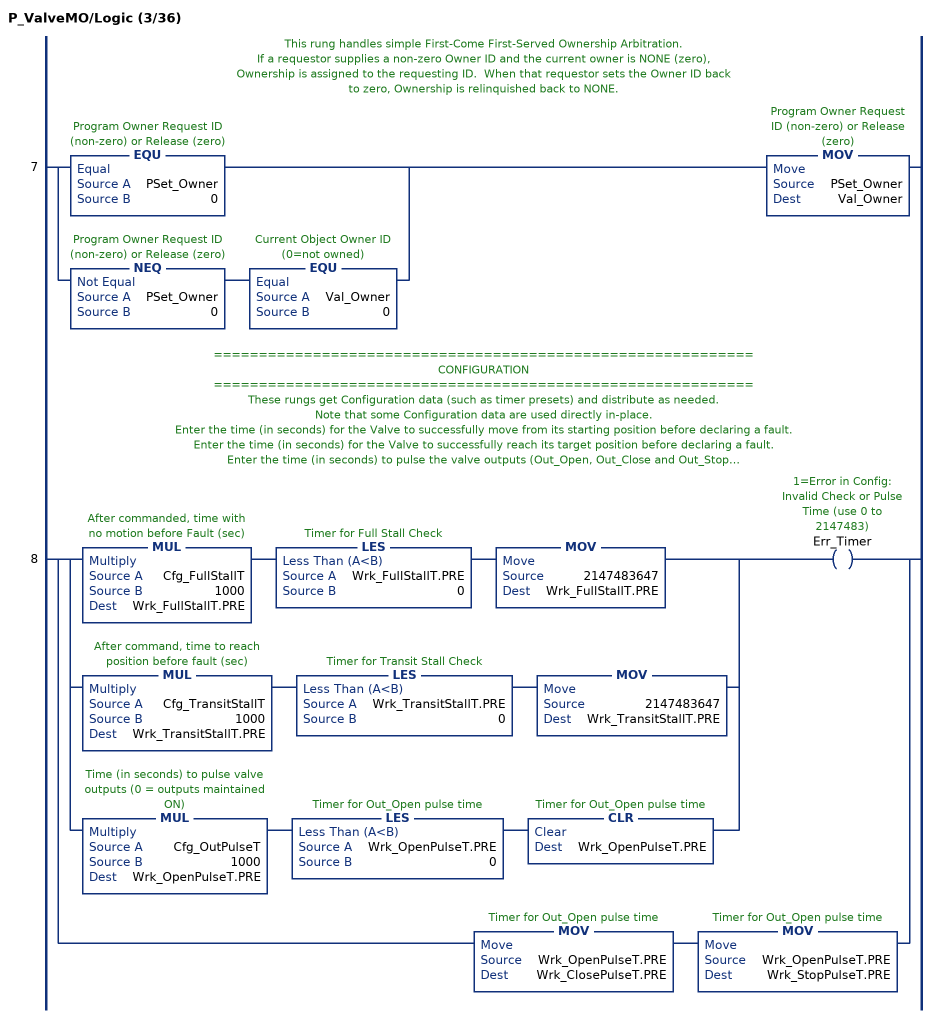
   // This rung handles simple First-Come First-Served Ownership Arbitration.
   // If a requestor supplies a non-zero Owner ID and the current owner is NONE (zero),
   // Ownership is assigned to the requesting ID.  When that requestor sets the Owner ID back
   // to zero, Ownership is relinquished back to NONE.
   7: [EQU(PSet_Owner,0) ,NEQ(PSet_Owner,0) EQU(Val_Owner,0) ]MOV(PSet_Owner,Val_Owner);
   // ============================================================
   // CONFIGURATION
   // ============================================================
   // These rungs get Configuration data (such as timer presets) and distribute as needed.
   // Note that some Configuration data are used directly in-place.
   // Enter the time (in seconds) for the Valve to successfully move from its starting position before declaring a fault.
   // Enter the time (in seconds) for the Valve to successfully reach its target position before declaring a fault.
   // Enter the time (in seconds) to pulse the valve outputs (Out_Open, Out_Close and Out_Stop)
   // (zero - held on continuously)
   // If the timer preset calcuated wraps negative (more than 2.14... million seconds), then max out the
   // Timer Preset.  Note that a negative timer preset will fault the controller!!!
   8: [[MUL(Cfg_FullStallT,1000,Wrk_FullStallT.PRE) LES(Wrk_FullStallT.PRE,0) MOV(2147483647,Wrk_FullStallT.PRE) ,MUL(Cfg_TransitStallT,1000,Wrk_TransitStallT.PRE) LES(Wrk_TransitStallT.PRE,0) MOV(2147483647,Wrk_TransitStallT.PRE) ,MUL(Cfg_OutPulseT,1000,Wrk_OpenPulseT.PRE) LES(Wrk_OpenPulseT.PRE,0) CLR(Wrk_OpenPulseT.PRE) ] OTE(Err_Timer) ,MOV(Wrk_OpenPulseT.PRE,Wrk_ClosePulseT.PRE) MOV(Wrk_OpenPulseT.PRE,Wrk_StopPulseT.PRE) ];
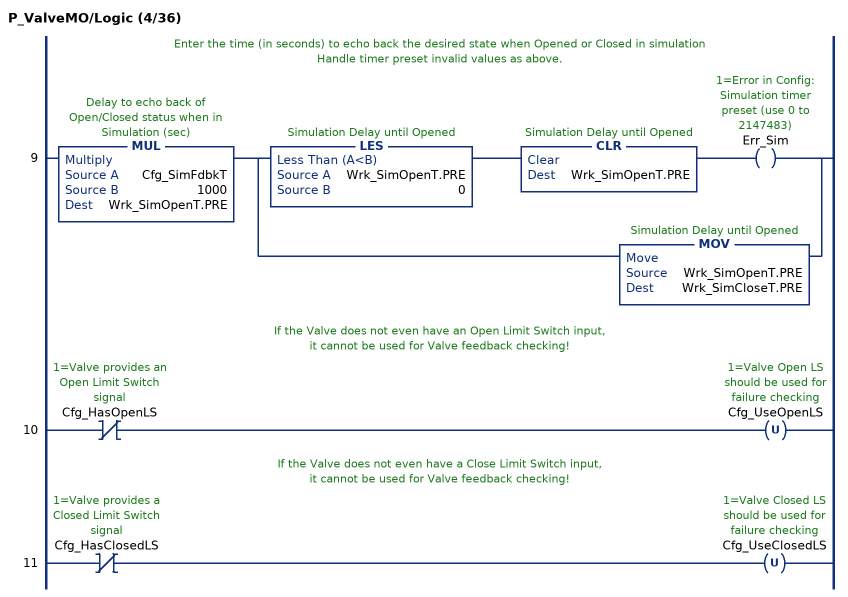
   // Enter the time (in seconds) to echo back the desired state when Opened or Closed in simulation
   // Handle timer preset invalid values as above.
   9: MUL(Cfg_SimFdbkT,1000,Wrk_SimOpenT.PRE)[LES(Wrk_SimOpenT.PRE,0) CLR(Wrk_SimOpenT.PRE) OTE(Err_Sim) ,MOV(Wrk_SimOpenT.PRE,Wrk_SimCloseT.PRE) ];
   // If the Valve does not even have an Open Limit Switch input,
   // it cannot be used for Valve feedback checking!
   10: XIO(Cfg_HasOpenLS)OTU(Cfg_UseOpenLS);
   // If the Valve does not even have a Close Limit Switch input,
   // it cannot be used for Valve feedback checking!
   11: XIO(Cfg_HasClosedLS)OTU(Cfg_UseClosedLS);
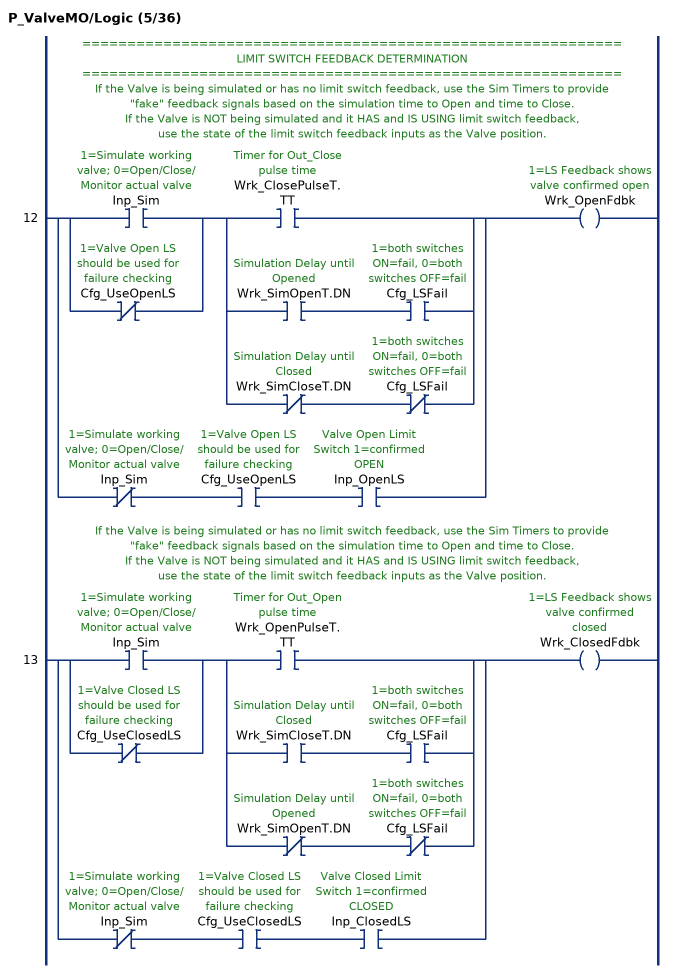
   // ============================================================
   // LIMIT SWITCH FEEDBACK DETERMINATION
   // ============================================================
   // If the Valve is being simulated or has no limit switch feedback, use the Sim Timers to provide
   // "fake" feedback signals based on the simulation time to Open and time to Close.
   // If the Valve is NOT being simulated and it HAS and IS USING limit switch feedback,
   // use the state of the limit switch feedback inputs as the Valve position.
   12: [[XIC(Inp_Sim) ,XIO(Cfg_UseOpenLS) ] [XIC(Wrk_ClosePulseT.TT) ,XIC(Wrk_SimOpenT.DN) XIC(Cfg_LSFail) ,XIO(Wrk_SimCloseT.DN) XIO(Cfg_LSFail) ] ,XIO(Inp_Sim) XIC(Cfg_UseOpenLS) XIC(Inp_OpenLS) ]OTE(Wrk_OpenFdbk);
   // If the Valve is being simulated or has no limit switch feedback, use the Sim Timers to provide
   // "fake" feedback signals based on the simulation time to Open and time to Close.
   // If the Valve is NOT being simulated and it HAS and IS USING limit switch feedback,
   // use the state of the limit switch feedback inputs as the Valve position.
   13: [[XIC(Inp_Sim) ,XIO(Cfg_UseClosedLS) ] [XIC(Wrk_OpenPulseT.TT) ,XIC(Wrk_SimCloseT.DN) XIC(Cfg_LSFail) ,XIO(Wrk_SimOpenT.DN) XIO(Cfg_LSFail) ] ,XIO(Inp_Sim) XIC(Cfg_UseClosedLS) XIC(Inp_ClosedLS) ]OTE(Wrk_ClosedFdbk);
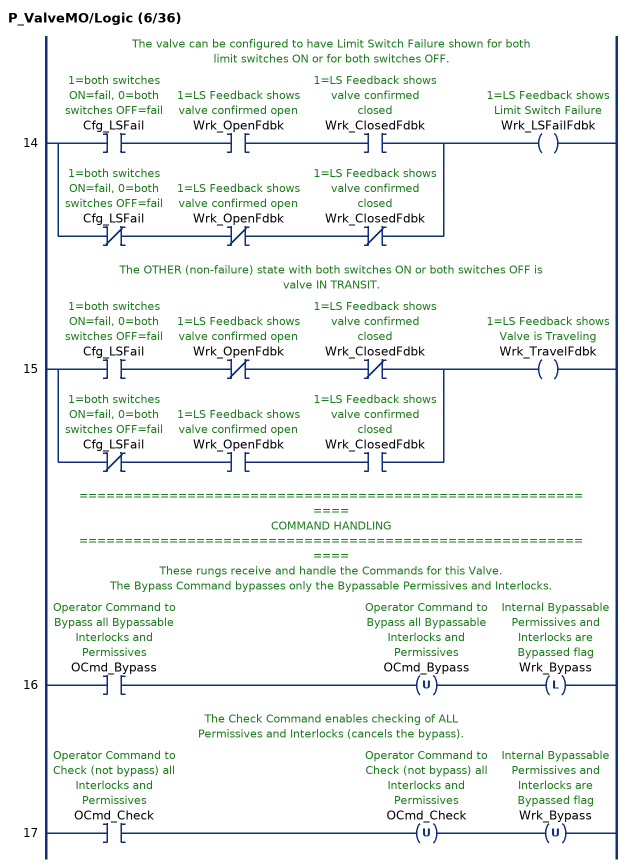
   // The valve can be configured to have Limit Switch Failure shown for both
   // limit switches ON or for both switches OFF.
   14: [XIC(Cfg_LSFail) XIC(Wrk_OpenFdbk) XIC(Wrk_ClosedFdbk) ,XIO(Cfg_LSFail) XIO(Wrk_OpenFdbk) XIO(Wrk_ClosedFdbk) ]OTE(Wrk_LSFailFdbk);
   // The OTHER (non-failure) state with both switches ON or both switches OFF is
   // valve IN TRANSIT.
   15: [XIC(Cfg_LSFail) XIO(Wrk_OpenFdbk) XIO(Wrk_ClosedFdbk) ,XIO(Cfg_LSFail) XIC(Wrk_OpenFdbk) XIC(Wrk_ClosedFdbk) ]OTE(Wrk_TravelFdbk);
   // ============================================================
   // COMMAND HANDLING
   // ============================================================
   // These rungs receive and handle the Commands for this Valve.
   // The Bypass Command bypasses only the Bypassable Permissives and Interlocks.
   16: XIC(OCmd_Bypass)OTU(OCmd_Bypass)OTL(Wrk_Bypass);
   // The Check Command enables checking of ALL
   // Permissives and Interlocks (cancels the bypass).
   17: XIC(OCmd_Check)OTU(OCmd_Check)OTU(Wrk_Bypass);
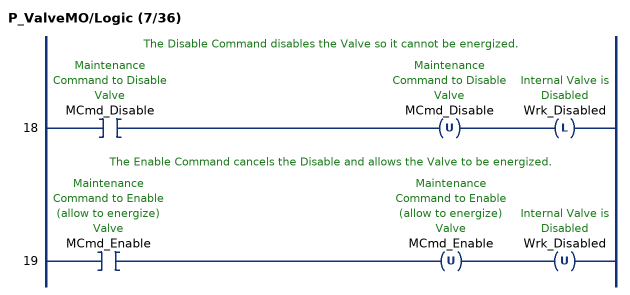
   // The Disable Command disables the Valve so it cannot be energized.
   18: XIC(MCmd_Disable)OTU(MCmd_Disable)OTL(Wrk_Disabled);
   // The Enable Command cancels the Disable and allows the Valve to be energized.
   19: XIC(MCmd_Enable)OTU(MCmd_Enable)OTU(Wrk_Disabled);
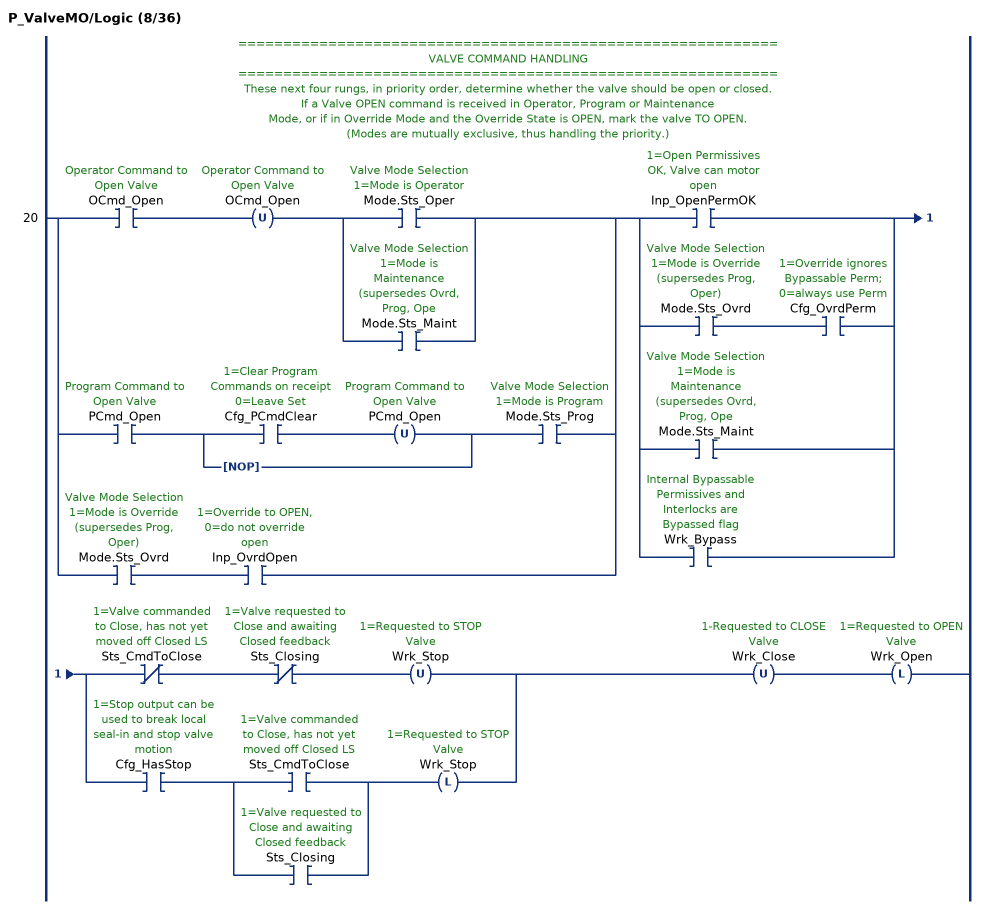
   // ============================================================
   // VALVE COMMAND HANDLING
   // ============================================================
   // These next four rungs, in priority order, determine whether the valve should be open or closed.
   // If a Valve OPEN command is received in Operator, Program or Maintenance
   // Mode, or if in Override Mode and the Override State is OPEN, mark the valve TO OPEN.
   // (Modes are mutually exclusive, thus handling the priority.)
   20: [XIC(OCmd_Open) OTU(OCmd_Open) [XIC(Mode.Sts_Oper) ,XIC(Mode.Sts_Maint) ] ,XIC(PCmd_Open) [XIC(Cfg_PCmdClear) OTU(PCmd_Open) ,NOP() ] XIC(Mode.Sts_Prog) ,XIC(Mode.Sts_Ovrd) XIC(Inp_OvrdOpen) ][XIC(Inp_OpenPermOK) ,XIC(Mode.Sts_Ovrd) XIC(Cfg_OvrdPerm) ,XIC(Mode.Sts_Maint) ,XIC(Wrk_Bypass) ][XIO(Sts_CmdToClose) XIO(Sts_Closing) OTU(Wrk_Stop) ,XIC(Cfg_HasStop) [XIC(Sts_CmdToClose) ,XIC(Sts_Closing) ] OTL(Wrk_Stop) ]OTU(Wrk_Close)OTL(Wrk_Open);
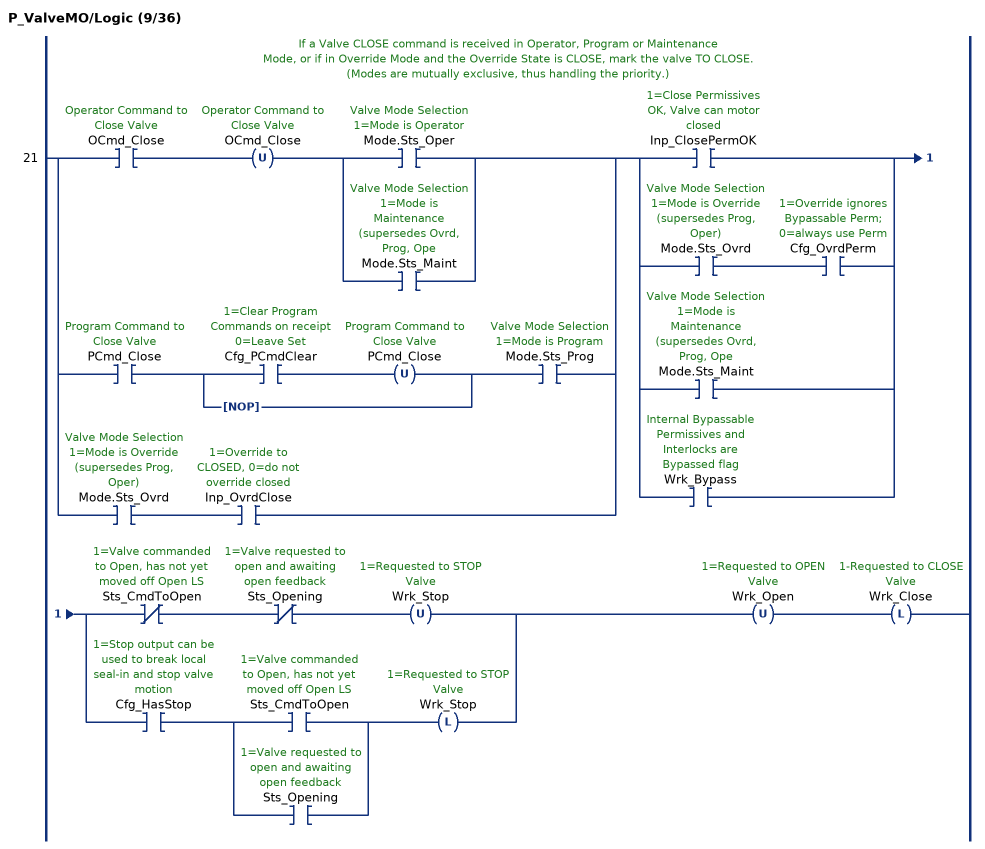
   // If a Valve CLOSE command is received in Operator, Program or Maintenance
   // Mode, or if in Override Mode and the Override State is CLOSE, mark the valve TO CLOSE.
   // (Modes are mutually exclusive, thus handling the priority.)
   21: [XIC(OCmd_Close) OTU(OCmd_Close) [XIC(Mode.Sts_Oper) ,XIC(Mode.Sts_Maint) ] ,XIC(PCmd_Close) [XIC(Cfg_PCmdClear) OTU(PCmd_Close) ,NOP() ] XIC(Mode.Sts_Prog) ,XIC(Mode.Sts_Ovrd) XIC(Inp_OvrdClose) ][XIC(Inp_ClosePermOK) ,XIC(Mode.Sts_Ovrd) XIC(Cfg_OvrdPerm) ,XIC(Mode.Sts_Maint) ,XIC(Wrk_Bypass) ][XIO(Sts_CmdToOpen) XIO(Sts_Opening) OTU(Wrk_Stop) ,XIC(Cfg_HasStop) [XIC(Sts_CmdToOpen) ,XIC(Sts_Opening) ] OTL(Wrk_Stop) ]OTU(Wrk_Open)OTL(Wrk_Close);
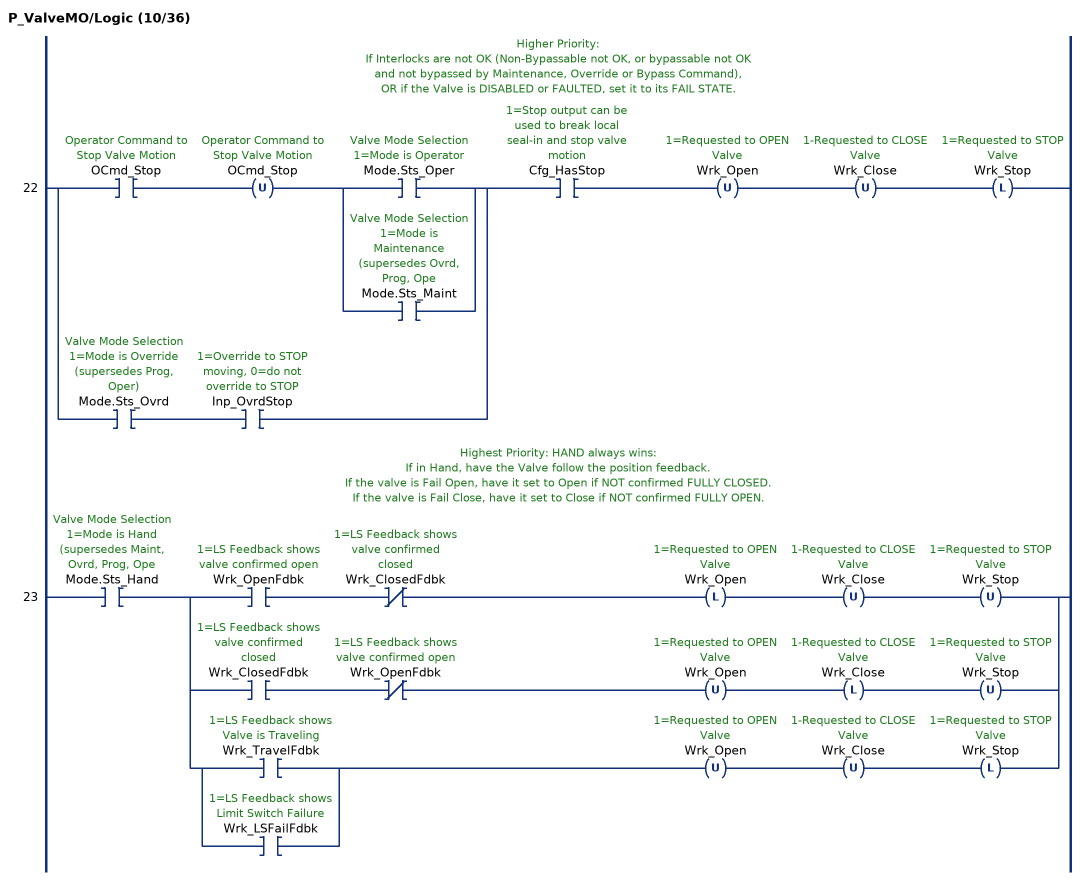
   // Higher Priority:
   // If Interlocks are not OK (Non-Bypassable not OK, or bypassable not OK
   // and not bypassed by Maintenance, Override or Bypass Command),
   // OR if the Valve is DISABLED or FAULTED, set it to its FAIL STATE.
   22: [XIC(OCmd_Stop) OTU(OCmd_Stop) [XIC(Mode.Sts_Oper) ,XIC(Mode.Sts_Maint) ] ,XIC(Mode.Sts_Ovrd) XIC(Inp_OvrdStop) ]XIC(Cfg_HasStop)OTU(Wrk_Open)OTU(Wrk_Close)OTL(Wrk_Stop);
   // Highest Priority: HAND always wins:
   // If in Hand, have the Valve follow the position feedback.
   // If the valve is Fail Open, have it set to Open if NOT confirmed FULLY CLOSED.
   // If the valve is Fail Close, have it set to Close if NOT confirmed FULLY OPEN.
   23: XIC(Mode.Sts_Hand)[XIC(Wrk_OpenFdbk) XIO(Wrk_ClosedFdbk) OTL(Wrk_Open) OTU(Wrk_Close) OTU(Wrk_Stop) ,XIC(Wrk_ClosedFdbk) XIO(Wrk_OpenFdbk) OTU(Wrk_Open) OTL(Wrk_Close) OTU(Wrk_Stop) ,[XIC(Wrk_TravelFdbk) ,XIC(Wrk_LSFailFdbk) ] OTU(Wrk_Open) OTU(Wrk_Close) OTL(Wrk_Stop) ];
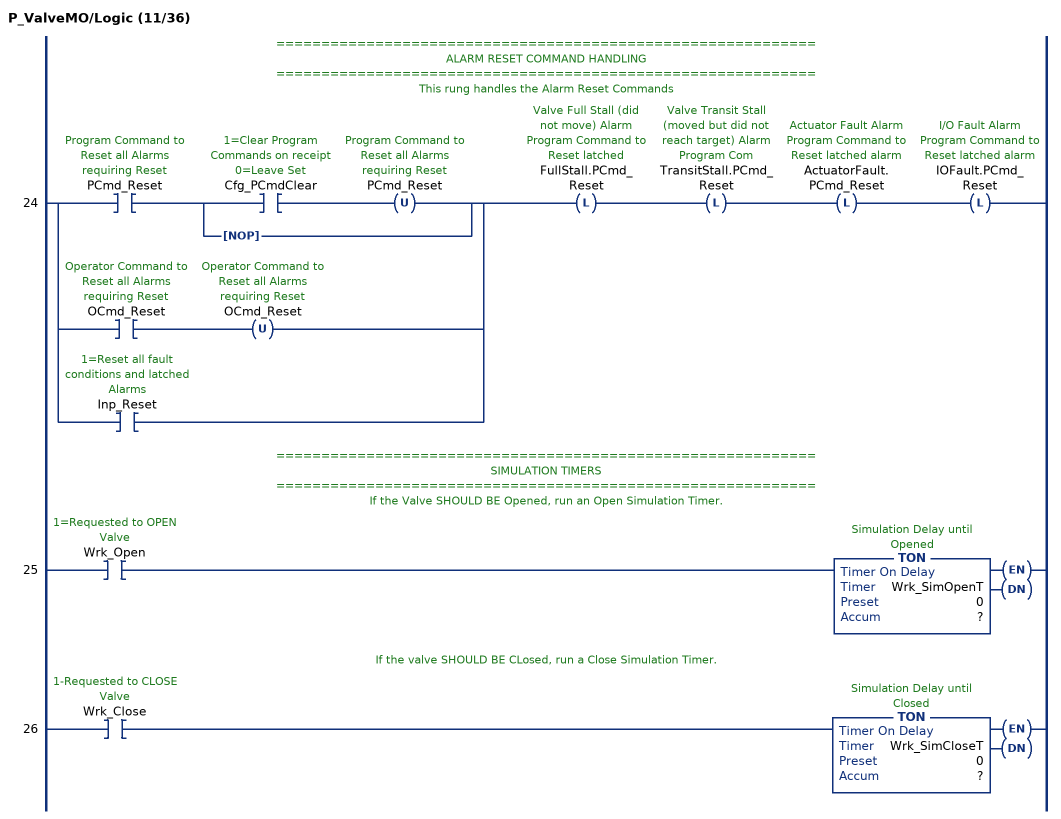
   // ============================================================
   // ALARM RESET COMMAND HANDLING
   // ============================================================
   // This rung handles the Alarm Reset Commands
   24: [XIC(PCmd_Reset) [XIC(Cfg_PCmdClear) OTU(PCmd_Reset) ,NOP() ] ,XIC(OCmd_Reset) OTU(OCmd_Reset) ,XIC(Inp_Reset) ]OTL(FullStall.PCmd_Reset)OTL(TransitStall.PCmd_Reset)OTL(ActuatorFault.PCmd_Reset)OTL(IOFault.PCmd_Reset);
   // ============================================================
   // SIMULATION TIMERS
   // ============================================================
   // If the Valve SHOULD BE Opened, run an Open Simulation Timer.
   25: XIC(Wrk_Open)TON(Wrk_SimOpenT,?,?);
   // If the valve SHOULD BE CLosed, run a Close Simulation Timer.
   26: XIC(Wrk_Close)TON(Wrk_SimCloseT,?,?);
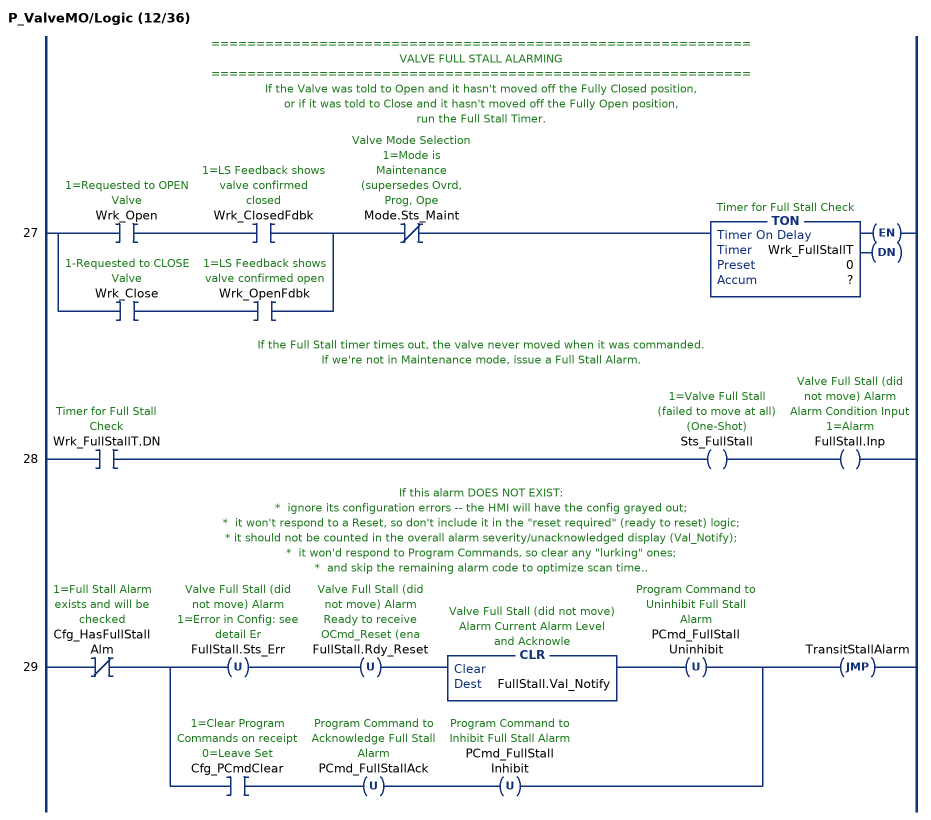
   // ============================================================
   // VALVE FULL STALL ALARMING
   // ============================================================
   // If the Valve was told to Open and it hasn't moved off the Fully Closed position,
   // or if it was told to Close and it hasn't moved off the Fully Open position,
   // run the Full Stall Timer.
   27: [XIC(Wrk_Open) XIC(Wrk_ClosedFdbk) ,XIC(Wrk_Close) XIC(Wrk_OpenFdbk) ]XIO(Mode.Sts_Maint)TON(Wrk_FullStallT,?,?);
   // If the Full Stall timer times out, the valve never moved when it was commanded.
   // If we're not in Maintenance mode, issue a Full Stall Alarm.
   28: XIC(Wrk_FullStallT.DN)OTE(Sts_FullStall)OTE(FullStall.Inp);
   // If this alarm DOES NOT EXIST:
   // *  ignore its configuration errors -- the HMI will have the config grayed out;
   // *  it won't respond to a Reset, so don't include it in the "reset required" (ready to reset) logic;
   // * it should not be counted in the overall alarm severity/unacknowledged display (Val_Notify);
   // *  it won'd respond to Program Commands, so clear any "lurking" ones;
   // *  and skip the remaining alarm code to optimize scan time..
   29: XIO(Cfg_HasFullStallAlm)[OTU(FullStall.Sts_Err) OTU(FullStall.Rdy_Reset) CLR(FullStall.Val_Notify) OTU(PCmd_FullStallUninhibit) ,XIC(Cfg_PCmdClear) OTU(PCmd_FullStallAck) OTU(PCmd_FullStallInhibit) ]JMP(TransitStallAlarm);
